DATA_BLOCK "DB"
{ S7_Optimized_Access := 'false' }
    VAR
        S1_vs1: DINT;
        S2_vs2: DINT;
        S2: DINT;
        R1_vr1: DINT;
        R2_vr2: DINT;
        R2: DINT;
        Y1_vy1: DINT;
        Y2_vy2: DINT;
        Y2: DINT;
        M1_vm1: DINT;
        M2_vm2: DINT;
        M2: DINT;
        firstRun: BOOL;
    END_VAR
BEGIN
    firstRun := TRUE;
END_DATA_BLOCK
